// This function has been automatically generated from the project information.
{attribute 'signature_flag' := '1073741824'}
{attribute 'TcGenerated'}
{attribute 'no-analysis'}
FUNCTION F_GetTitle : WSTRING
VAR_INPUT
	
END_VAR

F_GetTitle := "CNM_OpModeHandlingInterfaces";

END_FUNCTION

(* stored: Version 1.1.0.1
   POU F_GetTitle: Id {4358e55d-f5f8-4c4b-9d5f-22aa3538b14f}, SpecialFunc None *)
